{attribute 'qualified_only'}
VAR_GLOBAL	
	B1 AT %I*: BOOL; 	// Sensor Wagen Position
	B2 AT %I*: BOOL;	// Sensor Wagen Voll
	F1 AT %I*: BOOL; 	// Motorschutzschalter Förderband
	F2 AT %I*: BOOL;	// Motorschutzschalter Schneckenförderer	
	S1 AT %I*: BOOL;	// Taster "Aus"
	S2 AT %I*: BOOL;	// Taster "Ein"
	S3 AT %I*: BOOL;	// Not-Halt
	S4 AT %I*: BOOL;	// Taster "Quittieren"
END_VAR

(* stored: Version 1.1.0.1, ProductVersion 3.1.4024.4
   GVL SimDI: Id {c2d05302-d374-4f85-80dd-41006a3e3277} *)
